// TIA Portal V19 export
TYPE "UDT_AIN"
   STRUCT
      chn : Struct   // Channel
         "type" { S7_SetPoint := 'True'} : UInt := 0;   // Type of measurement: 0=hmi, 1=H-L, 2=factor
         in : Real := 0.0;   // Input to real number
         high { S7_SetPoint := 'True'} : Real := 0.0;   // Channel high limit (ex. 27648)
         low { S7_SetPoint := 'True'} : Real := 0.0;   // Channel high limit (ex. 0)
      END_STRUCT;
      scale : Struct   // Scaling
         high { S7_SetPoint := 'True'} : Real := 0.0;   // High limit of scale process
         low { S7_SetPoint := 'True'} : Real := 0.0;   // Low limit of scale process
         factor { S7_SetPoint := 'True'} : Real := 0.0;   // Factor multiplied to real number
         set : Bool := false;   // Scaling setup is complete
      END_STRUCT;
      sim : Struct   // Simulation
         en { S7_SetPoint := 'True'} : Bool := false;   // Simulation command
         value { S7_SetPoint := 'True'} : Real := 0.0;   // Simulation value
      END_STRUCT;
      exp : Struct   // Exponential filter
         en { S7_SetPoint := 'True'} : Bool := false;   // Exponential smoothing function (1=en, 0=dis)
         init : Bool := false;   // Exponential function initialized
         T { S7_SetPoint := 'True'} : Real := 0.0;   // Time to reach 63.2% = 1-1/e of original signal (must >=Dt)
         limit { S7_SetPoint := 'True'} : Real := 0.0;   // Limit near value that forces the Sn to break the loop and catch the Xn
         "dt" : Real := 0.0;   // Dt in ms
         "a" : Real := 0.0;   // a = 1- e^(-Dt/T) and if Dt<<<T then a=Dt/T
      END_STRUCT;
      faults : Struct   // Alarms
         hh { S7_SetPoint := 'True'} : "UDT_ALARMACKN";
         h { S7_SetPoint := 'True'} : "UDT_ALARMACKN";
         l { S7_SetPoint := 'True'} : "UDT_ALARMACKN";
         ll { S7_SetPoint := 'True'} : "UDT_ALARMACKN";
         sp_hh { S7_SetPoint := 'True'} : Real := 0.0;   // Setpoint of high-high alarm
         sp_h { S7_SetPoint := 'True'} : Real := 0.0;   // Setpoint of high alarm
         sp_l { S7_SetPoint := 'True'} : Real := 0.0;   // Setpoint of low alarm
         sp_ll { S7_SetPoint := 'True'} : Real := 0.0;   // Setpoint of low-low alarm
         fpreset : Bool := false;   // Reset Alarms
      END_STRUCT;
      trendlow { S7_SetPoint := 'True'} : Real := 0.0;   // Low limit of trend y axis = ymin - abs(ymax)*0.1
      trendhigh { S7_SetPoint := 'True'} : Real := 0.0;   // High limit of trend y axis = ymax + abs(ymax)*0.1
      scaled : Real := 0.0;   // Output value after scaling
      output : Real := 0.0;   // Output value after smoothing (or not if disabled)
      unit { S7_SetPoint := 'True'} : WString := WSTRING#'';   // Unit
   END_STRUCT;
END_TYPE
